FUNCTION ST08X_TO_BOOLS (* this Function extracts the 8 BOOLS from a 8-BOOL Struct *)
  (* Standard: 61499-1; Description: Copyright (c) 2024 HR Agrartechnik GmbH This program and the accompanying materials are made available under the terms of the Eclipse Public License 2.0 which is available at https://www.eclipse.org/legal/epl-2.0/ SPDX-License-Identifier: EPL-2.0 *)
  (* Version 1.0, 2024-02-22, Franz Höpfinger, HR Agrartechnik GmbH *)
  PACKAGE logiBUS::utils::conversion::str::forwarding;
  IMPORT eclipse4diac::core::TypeHash;
  IMPORT logiBUS::utils::conversion::types::ST08X;
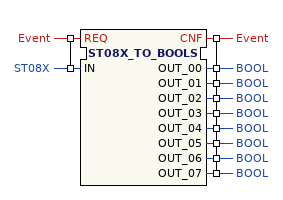
  EVENT_INPUT
    REQ WITH IN;
  END_EVENT
  EVENT_OUTPUT
    CNF WITH OUT_00, OUT_01, OUT_02, OUT_03, OUT_04, OUT_05, OUT_06, OUT_07;
  END_EVENT
  VAR_INPUT
    IN : logiBUS::utils::conversion::types::ST08X; (* ST08X Input *)
  END_VAR
  VAR_OUTPUT
    OUT_00 : BOOL; (* BIT 00 *)
    OUT_01 : BOOL; (* BIT 01 *)
    OUT_02 : BOOL; (* BIT 02 *)
    OUT_03 : BOOL; (* BIT 03 *)
    OUT_04 : BOOL; (* BIT 04 *)
    OUT_05 : BOOL; (* BIT 05 *)
    OUT_06 : BOOL; (* BIT 06 *)
    OUT_07 : BOOL; (* BIT 07 *)
  END_VAR
  BODY IN ST:
PACKAGE logiBUS::utils::conversion::str::forwarding;

IMPORT logiBUS::utils::conversion::types::ST08X;

(* this Function extracts the 8 BOOLS from a 8-BOOL Struct *)
FUNCTION ST08X_TO_BOOLS

VAR_INPUT
	IN : ST08X; // ST08X Input
END_VAR

VAR_OUTPUT
	OUT_00 : BOOL; // BIT 00
	OUT_01 : BOOL; // BIT 01
	OUT_02 : BOOL; // BIT 02
	OUT_03 : BOOL; // BIT 03
	OUT_04 : BOOL; // BIT 04
	OUT_05 : BOOL; // BIT 05
	OUT_06 : BOOL; // BIT 06
	OUT_07 : BOOL; // BIT 07
END_VAR

OUT_00 := IN.X_00;
OUT_01 := IN.X_01;
OUT_02 := IN.X_02;
OUT_03 := IN.X_03;
OUT_04 := IN.X_04;
OUT_05 := IN.X_05;
OUT_06 := IN.X_06;
OUT_07 := IN.X_07;

END_FUNCTION
  END_BODY
END_FUNCTION
